FUNCTION_BLOCK fb_V3BarcodeMasterCtrl
VAR_INPUT
	
	sBarcodeReceived								: STRING;
	b1stBasketMemoryFlag							: BOOL;
	bHandHeldBarcodeScannerEn 						: BOOL;
	bFixedTypeBarcodeScannerEn 						: BOOL;
	bON_ForHandHeldTypeOnly 						: BOOL;
	bON_ForFixedTypeOnly 							: BOOL;
	bStringEliminatorEn 								: BOOL;
	bBarcodeRegEn 									: BOOL;
	bScrollUpPB 										: BOOL;
	bScrollDownPB 									: BOOL;
	bTracerEn 										: BOOL;
	bfbV1_UTAC 										: BOOL;
	bfbV2 											: BOOL;
	iCharEliminateQty 									: INT;
	iCharNeededQty 									: INT;
(*
	ARsBarCodeRaw_V2 : ARRAY [0..99] OF STRING;
	ARsBarcodeDescrip_V2 : ARRAY [0..99] OF STRING;
*)

END_VAR

VAR_IN_OUT
END_VAR

VAR_OUTPUT
	bStringEliminatorDone 								: BOOL;
	bStringEliminatorError								: BOOL;
	bUpEndFlag 										: BOOL;
	bDownEndFlag 									: BOOL;
	bBarcodeTraceSuccess 							: BOOL;
	bBarcodeTraceFail 								: BOOL;
	iBarcodeRecipeNo_OUT 							: INT;
	sStringEliminatorStatus 							: STRING(50);
	sStringEliminatorResult 							: STRING;
	sBarcodeRegistrationStatus 						: STRING;
	sBarcodeDescrip_OUT 							: STRING;
(*
	sSendString						: STRING;
	sReceivedString					: STRING;
*)
END_VAR
VAR
	fbV3BarcodeScanner								: fb_V3BarcodeScanner;
	fbV3StringEliminator 								: fb_V3StringEliminator;
	fbV1BarcodeRegistration 							: fb_V1BarcodeRegistration_UTAC;
	fbV2BarcodeRegistration							: fb_V2BarcodeRegistration;
	fbV3BarcodeTracer 								: fb_V3BarcodeTracer;
	fbV3BarcodeRegSectionDisplayController 			: fb_V3BarcodeRegSectionDisplayController;

	sReceivedString									: STRING;

END_VAR
VAR // added by the converter: edge detectors and wires of the graphical bodies
    _w1 : STRING(INT#0);
END_VAR

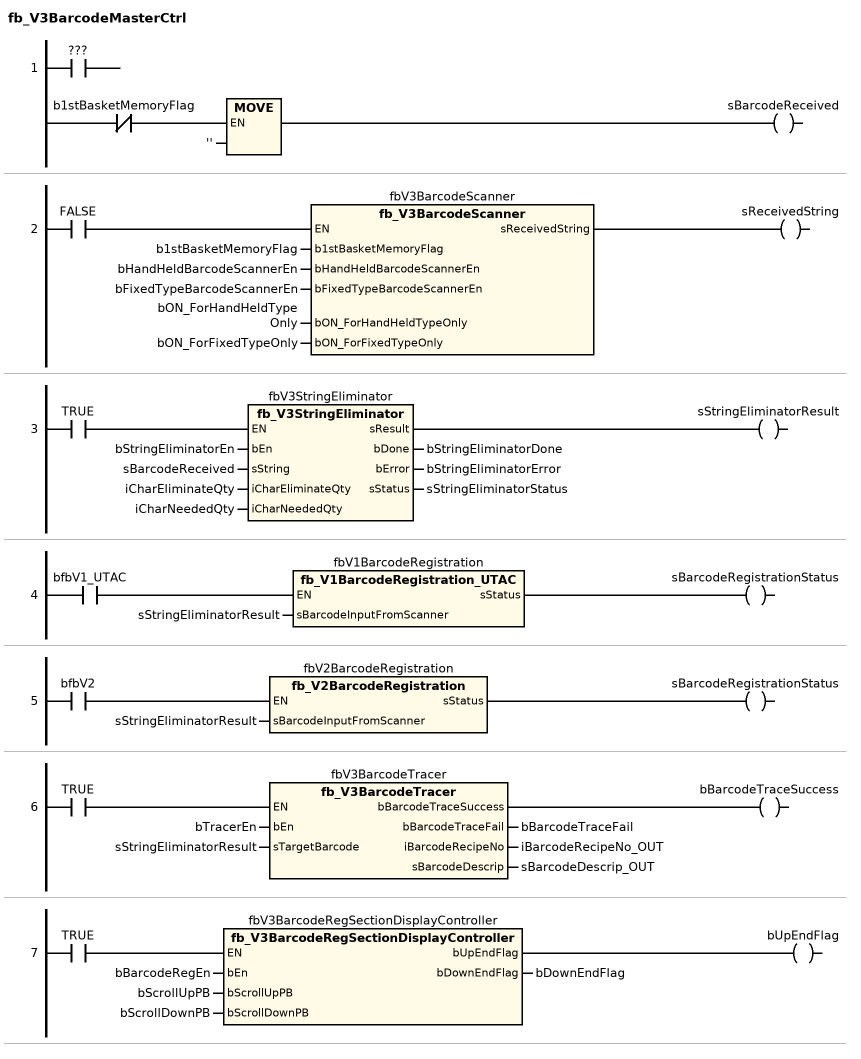
// NETWORK 1
IF NOT b1stBasketMemoryFlag THEN _w1 := ''; END_IF
sBarcodeReceived := _w1;

// NETWORK 2
IF FALSE THEN
    fbV3BarcodeScanner(
        b1stBasketMemoryFlag := b1stBasketMemoryFlag,
        bHandHeldBarcodeScannerEn := bHandHeldBarcodeScannerEn,
        bFixedTypeBarcodeScannerEn := bFixedTypeBarcodeScannerEn,
        bON_ForHandHeldTypeOnly := bON_ForHandHeldTypeOnly,
        bON_ForFixedTypeOnly := bON_ForFixedTypeOnly); // fb_V3BarcodeScanner
END_IF
sReceivedString := fbV3BarcodeScanner.sReceivedString;

// NETWORK 3
fbV3StringEliminator(
    bEn := bStringEliminatorEn,
    sString := sBarcodeReceived,
    iCharEliminateQty := iCharEliminateQty,
    iCharNeededQty := iCharNeededQty,
    bDone => bStringEliminatorDone,
    bError => bStringEliminatorError,
    sStatus => sStringEliminatorStatus); // fb_V3StringEliminator
sStringEliminatorResult := fbV3StringEliminator.sResult;

// NETWORK 4
IF bfbV1_UTAC THEN
    fbV1BarcodeRegistration(sBarcodeInputFromScanner := sStringEliminatorResult); // fb_V1BarcodeRegistration_UTAC
END_IF
sBarcodeRegistrationStatus := fbV1BarcodeRegistration.sStatus;

// NETWORK 5
IF bfbV2 THEN
    fbV2BarcodeRegistration(sBarcodeInputFromScanner := sStringEliminatorResult); // fb_V2BarcodeRegistration
END_IF
sBarcodeRegistrationStatus := fbV2BarcodeRegistration.sStatus;

// NETWORK 6
fbV3BarcodeTracer(
    bEn := bTracerEn,
    sTargetBarcode := sStringEliminatorResult,
    bBarcodeTraceFail => bBarcodeTraceFail,
    iBarcodeRecipeNo => iBarcodeRecipeNo_OUT,
    sBarcodeDescrip => sBarcodeDescrip_OUT); // fb_V3BarcodeTracer
bBarcodeTraceSuccess := fbV3BarcodeTracer.bBarcodeTraceSuccess;

// NETWORK 7
fbV3BarcodeRegSectionDisplayController(
    bEn := bBarcodeRegEn,
    bScrollUpPB := bScrollUpPB,
    bScrollDownPB := bScrollDownPB,
    bDownEndFlag => bDownEndFlag); // fb_V3BarcodeRegSectionDisplayController
bUpEndFlag := fbV3BarcodeRegSectionDisplayController.bUpEndFlag;

END_FUNCTION_BLOCK

(* stored: Version 1.1.0.1, ProductVersion 3.1.4024.12
   POU fb_V3BarcodeMasterCtrl: Id {a24200f5-29a6-43a4-9b75-32810ff643ab}, SpecialFunc None *)
